SUBAPPLICATION Uebung_012 (* Subapplication Type *)
  (* Standard: 61499-2 *)
  (* Version 1.0, 2023-10-23, franz *)
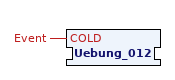
  EVENT_INPUT
    COLD;
  END_EVENT
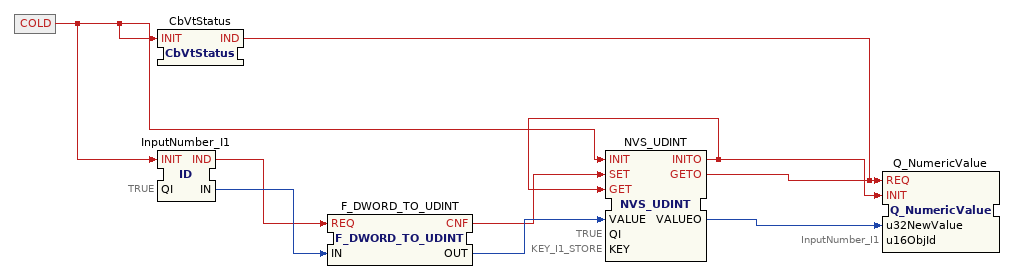
  FBS
    F_DWORD_TO_UDINT : F_DWORD_TO_UDINT;
    InputNumber_I1 : ID(QI := TRUE);
    NVS_UDINT : NVS_UDINT(QI := TRUE, KEY := KEY_I1_STORE);
    Q_NumericValue : Q_NumericValue(u16ObjId := InputNumber_I1);
    CbVtStatus : CbVtStatus;
  END_FBS
  EVENT_CONNECTIONS
    InputNumber_I1.IND TO F_DWORD_TO_UDINT.REQ;
    COLD TO InputNumber_I1.INIT;
    COLD TO NVS_UDINT.INIT;
    F_DWORD_TO_UDINT.CNF TO NVS_UDINT.SET;
    NVS_UDINT.INITO TO NVS_UDINT.GET;
    NVS_UDINT.GETO TO Q_NumericValue.REQ;
    NVS_UDINT.INITO TO Q_NumericValue.INIT;
    COLD TO CbVtStatus.INIT;
    CbVtStatus.IND TO Q_NumericValue.REQ;
  END_CONNECTIONS
  DATA_CONNECTIONS
    InputNumber_I1.IN TO F_DWORD_TO_UDINT.IN;
    F_DWORD_TO_UDINT.OUT TO NVS_UDINT.VALUE;
    NVS_UDINT.VALUEO TO Q_NumericValue.u32NewValue;
  END_CONNECTIONS
END_SUBAPPLICATION
